FUNCTION_BLOCK AX2_TO_AX (* Composite FB for convert bidirectional AX2 to unidirectional AX *)
  (* Standard: 61499-2; Function: AX2_BIDIR forwards its incoming (EO1) side out as a plain unidirectional signal via AX_OUT. AX_IN publishes its value onto the outgoing (EI1) side of AX2_BIDIR.; Description: Copyright (c) 2026 HR Agrartechnik GmbH This program and the accompanying materials are made available under the terms of the Eclipse Public License 2.0 which is available at https://www.eclipse.org/legal/epl-2.0/ SPDX-License-Identifier: EPL-2.0 *)
  (* Version 1.0, 2026-08-31, Franz Höpfinger, HR Agrartechnik GmbH, Initial Version *)
  PACKAGE adapter::conversion::bidirectional;
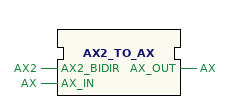
  SOCKETS
    AX2_BIDIR : adapter::types::bidirectional::AX2; (* Adapter Input: bidirectional tap, incoming side forwarded to AX_OUT, outgoing side driven by AX_IN *)
    AX_IN : adapter::types::unidirectional::AX; (* Adapter Input: unidirectional source *)
  END_SOCKETS
  PLUGS
    AX_OUT : adapter::types::unidirectional::AX; (* Adapter Output: mirrors AX2_BIDIR's incoming (indication) side *)
  END_PLUGS
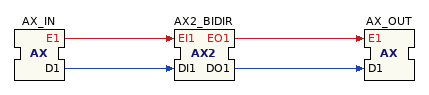
  EVENT_CONNECTIONS
    AX2_BIDIR.EO1 TO AX_OUT.E1;
    AX_IN.E1 TO AX2_BIDIR.EI1;
  END_CONNECTIONS
  DATA_CONNECTIONS
    AX2_BIDIR.DO1 TO AX_OUT.D1;
    AX_IN.D1 TO AX2_BIDIR.DI1;
  END_CONNECTIONS
END_FUNCTION_BLOCK
